PROGRAM MAIN
VAR

END_VAR

//Old
OOPSOld();

//Under Developement
OOPSDevelopmentTest();

END_PROGRAM

(* stored: Version 1.1.0.1, ProductVersion 3.1.4024.12
   POU MAIN: Id {75d8bf51-bd76-434e-a119-eb5787d14104}, SpecialFunc None *)
